{attribute 'linkalways'} 
{attribute 'no_explicit_call' := 'This FB is a CLASS and must be accessed using methods or properties'}
{attribute 'enable_dynamic_creation'}
FUNCTION_BLOCK _ETcVnOcrOptions EXTENDS EnumDatatypeBase
VAR
	localData : ETcVnOcrOptions;
	activeData : REFERENCE TO ETcVnOcrOptions;
	enumBaseDatatype : _UDINT(localData);
END_VAR

METHOD PRIVATE AddLocalEnumeration
VAR_INPUT
	Enumeration : T_MAXSTRING;
	Value : ETcVnOcrOptions;
END_VAR
AddEnumeration(Enumeration, Value);
END_METHOD

PROPERTY PUBLIC Address : PVOID
GET
Address := ADR(activeData);
END_GET
END_PROPERTY

METHOD PUBLIC ClearReference
VAR_INPUT
END_VAR
activeData REF= localData;
SetBaseDatatypeReference();
END_METHOD

METHOD PUBLIC Clone : I_Datatype
VAR
    pClone : POINTER TO _ETcVnOcrOptions;
END_VAR
pClone := __NEW(_ETcVnOcrOptions(InitialValue := Value));
Clone := pClone^;
END_METHOD

METHOD FB_init : BOOL
VAR_INPUT
	bInitRetains : BOOL; // if TRUE, the retain variables are initialized (warm start / cold start)
	bInCopyCode : BOOL;  // if TRUE, the instance afterwards gets moved into the copy code (online change)
	InitialValue : ETcVnOcrOptions;
END_VAR
localData := InitialValue;
AddBaseDatatype(enumBaseDatatype);
ClearReference();

AddLocalEnumeration('TCVN_OO_WITHBLANKS', ETcVnOcrOptions.TCVN_OO_WITHBLANKS);
END_METHOD

PROPERTY PUBLIC Identifier : T_MAXSTRING
GET
Identifier := 'ETcVnOcrOptions';
END_GET
END_PROPERTY

METHOD IsEnumeratorValueEqual : BOOL
VAR_INPUT
	Enumerator : I_KeyValueForwardEnumerator;
END_VAR
VAR
	storedValue : ETcVnOcrOptions;
END_VAR
IF NOT Enumerator.TryGet(storedValue) THEN
	RETURN;
END_IF

IsEnumeratorValueEqual := storedValue = activeData;
END_METHOD

METHOD PUBLIC MakeReferenceTo
VAR_INPUT
	ReferenceTarget : REFERENCE TO ETcVnOcrOptions;
END_VAR
activeData REF= ReferenceTarget;
SetBaseDatatypeReference();
END_METHOD

METHOD PROTECTED SetBaseDatatypeReference
VAR_INPUT
END_VAR
enumBaseDatatype.MakeReferenceTo(activeData);
END_METHOD

PROPERTY PUBLIC Size : UDINT
GET
Size := SIZEOF(activeData);
END_GET
END_PROPERTY

METHOD TryMakeReferenceTo : BOOL
VAR_INPUT
	Target : I_Datatype;
END_VAR
VAR
	targetAsEnum : I_EnumDatatype;
	pTargetData : POINTER TO ETcVnOcrOptions;
END_VAR
IF NOT Target.TryResolveAsEnumDatatype(targetAsEnum) THEN
	RETURN;
END_IF

IF targetAsEnum.Identifier <> Identifier THEN
	RETURN;
END_IF

pTargetData := Target.Address;
activeData REF= pTargetData^;
SetBaseDatatypeReference();
TryMakeReferenceTo := TRUE;
END_METHOD

PROPERTY PUBLIC Value : ETcVnOcrOptions
GET
Value := activeData;
END_GET
SET
activeData := Value;
END_SET
END_PROPERTY

END_FUNCTION_BLOCK

(* stored: Version 1.1.0.1
   POU _ETcVnOcrOptions: Id {799b6f0d-5ab6-470a-bb49-db6bfc083804}, SpecialFunc None
   Folder Constructor: Id {d48753aa-9c13-4fdd-ba8e-7fe8abe162d2}
   Folder Private: Id {f9d64c7b-18e2-48e3-84f2-e5f2f82fa968}
   Folder Protected: Id {e45513c0-748b-42c7-a92b-316b620d513d}
   Method AddLocalEnumeration: Id {0373a73c-5f2d-4101-bf10-d922a7906883}
   Property Address: Id {7706d080-fd28-4c68-a113-0b4e20d2621b}
   Get Get: Id {062ac5d4-a0fd-4468-b805-97a454aee3a5}
   Method ClearReference: Id {45b93017-f380-4d2d-b954-7f1cc468a6ca}
   Method Clone: Id {629e65c8-2912-4bbf-b295-1173a7239916}
   Method FB_init: Id {37387c68-d501-410d-8949-fdbbc9c1fd8a}
   Property Identifier: Id {e43340b1-5d82-4b48-b40b-7ab68f895fbb}
   Get Get: Id {be5eeac2-bcea-4cda-aa7c-b2ba2d0f8764}
   Method IsEnumeratorValueEqual: Id {d7005cf3-2350-40e7-a6b4-f2fd98fc09a7}
   Method MakeReferenceTo: Id {118900f7-9d0b-439f-8805-b1be15aa962d}
   Method SetBaseDatatypeReference: Id {2c54a346-9dc1-49d7-914a-b7417ae7bad6}
   Property Size: Id {9472e92b-8c70-4dbf-9873-8c3120096799}
   Get Get: Id {f0146566-7ab3-415e-b18e-dba0f2b2481c}
   Method TryMakeReferenceTo: Id {eebdaffa-37e2-4c43-9c2d-9206173a5ca0}
   Property Value: Id {f9f28eeb-abce-48d3-ac24-f13a912367c2}
   Get Get: Id {9955e093-fb59-42d9-8ab2-65fb8c86e1c5}
   Set Set: Id {13de478c-6b30-40e8-a0a9-03cb2bcd135b} *)
